Omron CX-Programmer project NewProject (CX-Programmer 9.75)

# PLC Memory_3: CP1E N30

## Program NewProgram1 (cyclic task 0)
Local symbols
M0 10.00 BOOL  ; 10.00
M1 10.01 BOOL  ; 10.01
M2 BOOL
M3 10.02 BOOL  ; 10.02
M4 10.03 BOOL  ; 10.03
M5 10.04 BOOL  ; 10.04
M6 10.05 BOOL  ; 10.05
Output 100.00 BOOL
PB 0.00 BOOL  ; 0.00
Reset 0.01 BOOL  ; 0.01

### Section Section1

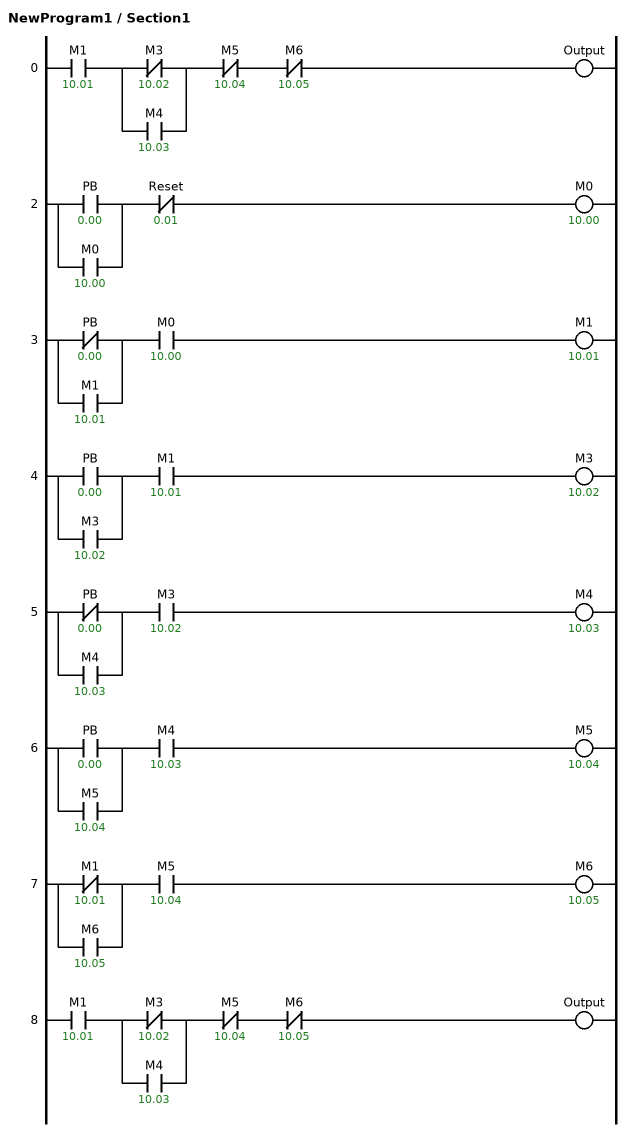
; rung 0
LD M1  ; 10.01
LDNOT M3  ; 10.02
OR M4  ; 10.03
ANDLD
ANDNOT M5  ; 10.04
ANDNOT M6  ; 10.05
OUT Output
; rung 2
LD PB  ; 0.00
OR M0  ; 10.00
ANDNOT Reset  ; 0.01
OUT M0  ; 10.00
; rung 3
LDNOT PB  ; 0.00
OR M1  ; 10.01
AND M0  ; 10.00
OUT M1  ; 10.01
; rung 4
LD PB  ; 0.00
OR M3  ; 10.02
AND M1  ; 10.01
OUT M3  ; 10.02
; rung 5
LDNOT PB  ; 0.00
OR M4  ; 10.03
AND M3  ; 10.02
OUT M4  ; 10.03
; rung 6
LD PB  ; 0.00
OR M5  ; 10.04
AND M4  ; 10.03
OUT M5  ; 10.04
; rung 7
LDNOT M1  ; 10.01
OR M6  ; 10.05
AND M5  ; 10.04
OUT M6  ; 10.05
; rung 8
LD M1  ; 10.01
LDNOT M3  ; 10.02
OR M4  ; 10.03
ANDLD
ANDNOT M5  ; 10.04
ANDNOT M6  ; 10.05
OUT Output

### Section END
; rung 0
END(001)